{attribute 'GeneratedUsingTerminal: EK1100-0000-0018'}
{attribute addProperty BoxType "EK1100-0000-0018"}
{attribute addProperty Id "Beckhoff_EP7xxxEK1122Beckhoff_EP7xxxEK1122_5EFC4D752992"}
{attribute addProperty CRC "3979743780"}
{attribute addProperty Size "2992"}
TYPE Beckhoff_EP7xxx_ED361224 EXTENDS EK1100_1FC0878B :
STRUCT
	{attribute addProperty Name "Beckhoff EP7xxxEK1122"}
	{attribute addProperty PreviousPort "Beckhoff EP7xxx : B"}
	Beckhoff_EP7xxxEK1122 : Beckhoff_EP7xxxEK1122_5EFC4D75;
END_STRUCT
END_TYPE

(* stored: Version 1.2.0.0, ProductVersion 3.1.4024.9
   DUT Beckhoff_EP7xxx_ED361224: Id {ca94e152-f1c0-44a3-ae48-f2381960cca2} *)
